(* CODESYS project ForOPC.export

Project tree, tasks and I/O mapping:
  application Application
    libraries: ; WagoAppStepper, 1.6.1.1 (WAGO)
    task PLC_Task (cyclic, interval t#50ms, priority 15) calls PLC_PRG
    DataTypes/
      data type CurveStates
      data type ForceStepStates
      data type StepperStates
      data type StiffnessTestStates
    GV/
      global variables AI_Sensors
      global variables HMI_Alm
      global variables HMI_Process
      global variables HMI_Stepper
    Program/
      Device/
        Motors/
          ForceStep/
            function block fbForceStep [ST]: METH_Direction
            program prForceStep [ST]
          Stepper/
            function block fbStepper [ST]: ACT_MoveHome, ACT_MoveToPos, METH_Direction
            program prLaserStepper_1 [ST]
            program prLaserStepper_2 [ST]
          program prMotion [ST]
        program prDevice [ST]
      IO/
        program prInToVars [ST]
      Process/
        GetCurve/
          function block fbGetCurve [ST]
          program prGetCurve_1 [ST]
          program prGetCurve_2 [ST]
        StiffnessTest/
          function block fbStiffnessTest [ST]
          program prStiffnessTest_1 [ST]
          program prStiffnessTest_2 [ST]
        program prProcess [ST]
      program prSimulation [ST]
    program PLC_PRG [ST]
    Symbols
*)

// Application/DataTypes/CurveStates

TYPE CurveStates :
(
	CS_Stop 		:= 0,
	CS_Done			:= 1,
	CS_Stopping		:= 2,
	CS_SetStep		:= 3,
	CS_WaitInitial	:= 4,
	CS_SetMeassure	:= 5,
	CS_Measuring	:= 6
);
END_TYPE

// Application/DataTypes/ForceStepStates

TYPE ForceStepStates :
(
	FS_Stop 				:= 0,
	FS_FirstRun 			:= 1,
	FS_WaitRaughApprox		:= 2,
	FS_MakeStep				:= 3,
	FS_CheckForce			:= 4,
	FS_Done					:= 5,
	FS_StartRelease			:= 6,
	FS_WaitRelease			:= 7,
	FS_MovePos				:= 8,
	FS_WaitVelicity			:= 9,
	FS_VelicityMode			:= 10,
	FS_VelicityStopping		:= 11
);
END_TYPE

// Application/DataTypes/StepperStates

TYPE StepperStates :
(
	SM_Idle 			:=0,
	SM_Homing			:=1,
	SM_Home				:=2,
	SM_SetPrm			:=3,
	SM_MovingToPos		:=4,
	SM_OnPos			:=5,
	SM_Stopping 		:=6,
	SM_Stop 			:=7
);
END_TYPE

// Application/DataTypes/StiffnessTestStates

TYPE StiffnessTestStates :
(
	ST_Proc_Stop 			:= 0,
	ST_Proc_GettingForce 	:= 1,
	ST_Proc_GettingHalfKoef	:= 2,
	ST_Proc_CalcKoef		:= 3,
	ST_Proc_GettingCurve	:= 4,
	ST_Proc_Done			:= 5,
	ST_Proc_Releasing		:= 6,
	ST_Proc_Stopping		:= 7
	
);
END_TYPE

// Application/GV/AI_Sensors

VAR_GLOBAL
	AI_Rol_1 		AT %IW1 : WORD;
	AI_Rol_2 		AT %IW2 : WORD;
	AI_Laser_1 		AT %IW3 : WORD;
	AI_Laser_2 		AT %IW4 : WORD;
	
	wCounter_1		AT %IW28 : WORD;
	wCounter_2		AT %IW30 : WORD;
	dwCounter		: DWORD;
END_VAR

// Application/GV/HMI_Alm

VAR_GLOBAL
	xResetAlm		: BOOL;
END_VAR

// Application/GV/HMI_Process

VAR_GLOBAL
	///////////////////////////   GET CURVE 1  //////////////////////
	
	xGC_Start_1: BOOL;
	wGS_State_1: CurveStates;
	
	///////////////////////////   GET CURVE 2  //////////////////////
	
	xGC_Start_2: BOOL;
	wGS_State_2: CurveStates;
	
	////////////////////////////  STIFFNESS TEST 1 /////////////////////////////
	
	xGS_StartProc_1: BOOL;
	wST_State_1: StiffnessTestStates;
	rST_Koef_1: REAL;
	wST_HalfPos_1: REAL;
	wST_HalfForce_1: REAL;
	xST_Ready_1: BOOL;
	
	////////////////////////////  STIFFNESS TEST 2 /////////////////////////////
	
	xGS_StartProc_2: BOOL;
	wST_State_2: StiffnessTestStates;
	rST_Koef_2: REAL;
	wST_HalfPos_2: REAL;
	wST_HalfForce_2: REAL;
	xST_Ready_2: BOOL;
	
	////////////////////////////  STIFFNESS TEST 3 /////////////////////////////
	
	xGS_StartProc_3: BOOL;
	wST_State_3: StiffnessTestStates;
	rST_Koef_3: REAL;
	wST_HalfPos_3: REAL;
	wST_HalfForce_3: REAL;
	xST_Ready_3: BOOL;
	
	////////////////////////////  DISTANCE /////////////////////////////
	
	rDistance_1		: REAL;
	rDistance_2		: REAL;
	rLaserDistance_1		: REAL;
	rLaserDistance_2		: REAL;
	
	xProcFinished			: BOOL;
	wProcType	: WORD;
	
END_VAR
VAR_GLOBAL RETAIN
	///////////////////////////   GET CURVE 1  //////////////////////
	
	wGC_Distance_1: WORD;
	wGC_InitialPos_1: WORD;
	wGC_EndPos_1: WORD;
	
	///////////////////////////   GET CURVE 2  //////////////////////
	
	wGC_Distance_2: WORD;
	wGC_InitialPos_2: WORD;
	wGC_EndPos_2: WORD;
	
	////////////////////////////  STIFFNESS TEST 1 /////////////////////////////
	
	rST_GetForce_1: REAL;
	rST_SetForce_1: REAL;
	wGS_WaitTillDone_1: WORD;
	
	////////////////////////////  STIFFNESS TEST 2 /////////////////////////////
	
	rST_GetForce_2: REAL;
	rST_SetForce_2: REAL;
	wGS_WaitTillDone_2: WORD;
	
END_VAR

// Application/GV/HMI_Stepper

VAR_GLOBAL
	///////////////////////    FORCE STEP    //////////////////////////////
	rFS_GetForce: REAL;	
	xFS_Start: BOOL;
	xFS_Release: BOOL;
	wFS_State: WORD;
	wFS_ActualPos: DWORD;
	xFS_JogLeft: BOOL;
	xFS_JogRight: BOOL;
	rFS_GetForce_check: REAL;	
	rFS_CycledWay:	REAL;
	rFS_LinedWay_1:	REAL;
	rFS_LinedWay_2:	REAL;
	
	
	///////////////////////////   LASER  STEP 1  //////////////////////
	xLS_MoveToPos_1: BOOL;
	xLS_MoveHome_1: BOOL;
	xLS_Stop_1: BOOL;
	wLS_GetPos_1: DINT;
	wLS_StepperState_1: WORD;
	xLS_Initilized_1: BOOL;
	rLS_RealPos_1:	REAL;
	
	///////////////////////////   LASER  STEP 2  //////////////////////
	xLS_MoveToPos_2: BOOL;
	xLS_MoveHome_2: BOOL;
	xLS_Stop_2: BOOL;
	wLS_GetPos_2: DINT;
	wLS_StepperState_2: WORD;
	xLS_Initilized_2: BOOL;
	rLS_RealPos_2:	REAL;
	
	
	
END_VAR
VAR_GLOBAL RETAIN
	
///////////////////////    FORCE STEP    //////////////////////////////
	rFS_SetForce: REAL;
	wFS_RoughApprox: WORD;
	wFS_Step: WORD;
	xFS_DirNeg: BOOL;
	rFS_Sensativity: REAL;
	wFS_SetSpeed: WORD;
	wFS_SetAcceleration: WORD;
	wFS_SetDeceleration: WORD;
	
	
///////////////////////////   LASER  STEP 1  //////////////////////	
	wLS_SetPos_1: WORD;
	wLS_SetSpeed_1: WORD;
	xLS_DirNeg_1: BOOL;
	wLS_Acceleration_1: WORD;
	wLS_Deceleration_1: WORD;
	
	///////////////////////////   LASER  STEP 2  //////////////////////	
	wLS_SetPos_2: WORD;
	wLS_SetSpeed_2: WORD;
	xLS_DirNeg_2: BOOL;
	wLS_Acceleration_2: WORD;
	wLS_Deceleration_2: WORD;
	
	
	
END_VAR

// Application/PLC_PRG
PROGRAM PLC_PRG
VAR
END_VAR

prDevice();
prProcess();
prSimulation();

END_PROGRAM

// Application/Program/Device/prDevice
PROGRAM prDevice
VAR
END_VAR

prMotion();

END_PROGRAM

// Application/Program/Device/Motors/prMotion
PROGRAM prMotion
VAR
END_VAR

prForceStep();
(*prLaserStepper_1();
prLaserStepper_2();*)

END_PROGRAM

// Application/Program/Device/Motors/ForceStep/prForceStep
PROGRAM prForceStep
VAR
	ForceStep:		fbForceStep;
	
	
	
END_VAR

ForceStep(
	rSetForce:= rFS_SetForce, 
	rGetForce:= rFS_GetForce, 
	wRoughApprox:= wFS_RoughApprox, 
	wStep:= wFS_Step, 
	xDirNeg:= xFS_DirNeg, 
	rSensativity:= rFS_Sensativity, 
	wSpeed:= wFS_SetSpeed, 
	wAcceleration:= wFS_SetAcceleration, 
	wDeceleration:= wFS_SetDeceleration, 
	I_Port:= IoConfig_Globals.Servo_Stepper_Controller_55_VDC_7_5A, 
	xStart:= xFS_Start, 
	xResetErr:= xResetAlm, 
	xRelease:= xFS_Release,
	xJogLeft:= xFS_JogLeft, 
	xJogRight:= xFS_JogRight,
	wState=> wFS_State, 
	diActualPosition=> );
	
	wFS_ActualPos:= ForceStep.diActualPosition;

END_PROGRAM

// Application/Program/Device/Motors/ForceStep/fbForceStep
FUNCTION_BLOCK fbForceStep
VAR_INPUT
	rSetForce:			REAL;
	rSetPos:			DINT;
	rGetForce:			REAL;
	wRoughApprox:		WORD;
	wStep:				WORD;
	xDirNeg:			BOOL;
	rSensativity:		REAL;
	wSpeed: 			WORD;
	wAcceleration: 		WORD;
	wDeceleration: 		WORD;
	I_Port: 			WagoAppStepper.WagoTypesModule_75x_67x.I_Module_75x_67x;
END_VAR
VAR_IN_OUT
	xStart:				BOOL;
	xResetErr:			BOOL;
	xRelease:			BOOL;
	xJogLeft:			BOOL;
	xJogRight:			BOOL;
END_VAR
VAR_OUTPUT
	wState:				ForceStepStates;
	diActualPosition: 	DINT;
END_VAR
VAR
	rtStart:			R_TRIG;
	ftStart:			F_TRIG;
	ftRelease:			F_TRIG;
	ControlBasic:		WagoAppStepper.FbStepperControlBasic;
	xEnable: 			BOOL;
	eJobType: 			WagoAppStepper.eMode;
	xTriggerStart: 		BOOL;
	xTriggerErrorReset: BOOL;
	xStop: 				BOOL;
	
	
	diPosition: 		DINT;
	iSpeed: 			INT;
	xJobFinished: 		BOOL;
	xBusy: 				BOOL;
	xError: 			BOOL;
	oStatus: 			WagoAppStepper.WagoSysErrorBase.FbResult;
	eErrorCodes: 		WagoAppStepper.eStatus;
	diRoughDistance:	DINT;
	rCompareForce:		REAL;
	rDirection:			INT;
	rtRelease:			R_TRIG;
	rtJogLeft:			R_TRIG;
	rtJogright:			R_TRIG;
	
END_VAR

VAR RETAIN
	diRetainPos: DINT;
END_VAR

rtStart(CLK:=xStart);
ftStart(CLK:=xStart);
rtRelease(CLK:=xRelease);
ftRelease(CLK:=xRelease);
rtJogLeft(CLK:=xJogLeft);
rtJogright(CLK:=xJogRight);

IF (ftStart.Q OR ftRelease.Q)AND (NOT (wState = FS_Done)) THEN
	xStop			:= TRUE;
	xTriggerStart	:= FALSE;
	xRelease		:= FALSE;	
	wState:=FS_Stop;
END_IF

IF rtRelease.Q THEN
	xStop			:=TRUE;
	xTriggerStart	:= FALSE;
	xJogLeft		:= FALSE;
	xJogRight		:= FALSE;
	wState			:=FS_StartRelease;
END_IF

IF (rtJogLeft.Q OR rtJogright.Q) AND (NOT(wState = FS_Stop OR wState = FS_Done)) THEN
	xJogLeft		:= FALSE;
	xJogRight		:= FALSE;
END_IF


CASE wState OF
	
		FS_Stop, FS_Done:
		
		
				IF rtStart.Q THEN
					diRoughDistance		:= 0;
					xStop				:=FALSE;
					rCompareForce		:= (rSetForce/100)* wRoughApprox;
					METH_Direction(xDirNeg:= xDirNeg);
					IF rSetPos = 0 THEN
						wState			:= FS_FirstRun;
					ELSE
						xEnable			:= TRUE;
						eJobType		:= MoveRelative;
						diPosition		:= rSetPos;
						iSpeed			:= wSpeed;
						xTriggerStart	:= TRUE;
						wState			:= FS_MovePos;
					END_IF					
				END_IF
				
				IF xJogLeft OR xJogRight THEN
					xEnable			:= TRUE;
					xStop			:=FALSE;
					eJobType		:= VelocityControl;
					METH_Direction(xDirNeg:= xJogLeft);
					iSpeed			:= (TO_INT(wSpeed)) * rDirection;
					xTriggerStart	:= TRUE;
					wState			:= FS_WaitVelicity;
				END_IF
					
		
		FS_FirstRun:
		
				xEnable			:= TRUE;
				eJobType		:= MoveRelative;
				diPosition		:= 200000 * rDirection;
				iSpeed			:= wSpeed;
				xTriggerStart	:=TRUE;
				wState			:= FS_WaitRaughApprox;
				
				
		FS_WaitRaughApprox:
		
				IF rGetForce > rCompareForce THEN
					xStop	:=TRUE;
					wState	:= FS_MakeStep;
				END_IF
				
		
		FS_MakeStep:
				
		
				IF xJobFinished THEN
					xStop			:=FALSE;
					diPosition		:= wStep * rDirection;
					xTriggerStart	:=TRUE;
					wState			:= FS_CheckForce;
				END_IF
				
				
		FS_CheckForce:
		
				
				IF xJobFinished THEN
					IF (rGetForce < rSetForce + rSensativity) AND (rGetForce > rSetForce - rSensativity) THEN
						xStart	:=FALSE;
						wState	:= FS_Done;
					ELSIF rGetForce < rSetForce - rSensativity THEN
						METH_Direction(xDirNeg:= xDirNeg);
						wState	:= FS_MakeStep;
					ELSIF rGetForce > rSetForce + rSensativity THEN
						METH_Direction(xDirNeg:= NOT xDirNeg);
						wState	:= FS_MakeStep;
					END_IF
				END_IF
				
		FS_StartRelease:
		
				IF xJobFinished THEN
					xStop			:=FALSE;
					METH_Direction(xDirNeg:= NOT xDirNeg);
					xEnable			:= TRUE;
					eJobType		:= MoveRelative;
					diPosition		:= 200000 * rDirection;
					iSpeed			:= wSpeed;
					xTriggerStart	:=TRUE;
					wState			:= FS_WaitRelease;
				END_IF
				
		FS_WaitRelease:
		
				IF rGetForce < rSensativity THEN
					xStart:= FALSE;
					xStop			:= TRUE;
					xTriggerStart	:= FALSE;
					xRelease		:= FALSE;	
					wState:=FS_Stop;
				END_IF
				
				
		FS_MovePos:
		
				IF xJobFinished THEN
					wState	:= FS_Done;
				END_IF
				
				
		FS_WaitVelicity:
		
				IF NOT xTriggerStart THEN
					wState	:= FS_VelicityMode;
				END_IF
				
				
		FS_VelicityMode:
		
		
				IF rtJogLeft.Q OR rtJogright.Q THEN
					xJogRight		:=rtJogright.Q;
					xJogLeft		:=rtJogLeft.Q;
					METH_Direction(xDirNeg:= xJogLeft);
					iSpeed			:= (TO_INT(wSpeed)) * rDirection;
					xTriggerStart	:= TRUE;
				END_IF
		
				IF NOT (xJogLeft OR xJogRight) THEN
					iSpeed			:= 0;
					xTriggerStart	:= TRUE;
					wState			:= FS_VelicityStopping;
				END_IF
				
				
		FS_VelicityStopping:
		
				IF ControlBasic.iActualSpeed = 0 AND (NOT xTriggerStart) THEN
					wState			:= FS_Stop;
				END_IF
				

END_CASE





ControlBasic(
	xEnable:= xEnable, 
	I_Port:= I_Port, 
	eJobType:= eJobType, 
	xDirPos:= NOT xDirNeg, 
	xDirNeg:= xDirNeg, 
	iSpeed:= iSpeed, 
	wAcceleration:= wAcceleration, 
	wDeceleration:= wDeceleration, 
	diPosition:= diPosition, 
	xTriggerStart:= xTriggerStart, 
	xTriggerErrorReset:= xTriggerErrorReset, 
	xStop:= xStop, 
	xJobFinished=> xJobFinished, 
	xBusy=> xBusy, 
	xError=> xError, 
	oStatus=> oStatus, 
	eErrorCodes=> eErrorCodes, 
	diActualPosition=> diActualPosition, 
	iActualSpeed=> , 
	xMailboxActive=> , 
	xResetWarning=> );

METHOD METH_Direction
VAR_INPUT
	xDirNeg:	BOOL;
END_VAR
IF xDirNeg THEN
	rDirection:= -1;
ELSE
	rDirection:= 1;
END_IF
END_METHOD

END_FUNCTION_BLOCK

// Application/Program/Device/Motors/Stepper/prLaserStepper_1
PROGRAM prLaserStepper_1
VAR
	LaserStepper	:	fbStepper;
	xMoveRelative	: 	BOOL;
	wRatio			: 	WORD:=10;
	
		
END_VAR

LaserStepper(
	diSetPos:= wLS_SetPos_1 * wRatio, 
	xMoveRelative:= xMoveRelative, 
	iSetSpeed:= wLS_SetSpeed_1 * wRatio, 
	xDirNeg:= xLS_DirNeg_1, 
	wAcceleration:= wLS_Acceleration_1, 
	wDeceleration:= wLS_Deceleration_1, 
	I_Port:= IoConfig_Globals.Servo_Stepper_Controller_55_VDC_7_5A_1, 
	xMoveToPos:= xLS_MoveToPos_1, 
	xMoveHome:= xLS_MoveHome_1, 
	xStop:= xLS_Stop_1, 
	diGetPos=> , 
	xInitilized=> xLS_Initilized_1, 
	wStepperState=> wLS_StepperState_1);
	
	wLS_GetPos_1:=LaserStepper.diGetPos/wRatio;

END_PROGRAM

// Application/Program/Device/Motors/Stepper/fbStepper
FUNCTION_BLOCK fbStepper
VAR_INPUT
	diSetPos:			DINT;
	xMoveRelative:		BOOL;
	iSetSpeed:			INT;
	xDirNeg:			BOOL;
	wAcceleration: 		WORD;
	wDeceleration: 		WORD;
	I_Port: 			WagoAppStepper.WagoTypesModule_75x_67x.I_Module_75x_67x;
END_VAR
VAR_IN_OUT
	xMoveToPos:			BOOL;
	xMoveHome:			BOOL;
	xStop:				BOOL;
END_VAR
VAR_OUTPUT
	diGetPos:			DINT;
	xInitilized:		BOOL;
	wStepperState:		StepperStates;
END_VAR
VAR
	rtMoveToPos:		R_TRIG;
	rtMoveHome:			R_TRIG;
	rtStop:				R_TRIG;
	ControlBasic:		WagoAppStepper.FbStepperControlBasic;
	xEnable: 			BOOL;
	eJobType: 			WagoAppStepper.eMode;
	xTriggerStart: 		BOOL;
	xTriggerErrorReset: BOOL;
	iSpeed: 			INT;
	
	diPosition: 		DINT;
	
	xJobFinished: 		BOOL;
	xBusy: 				BOOL;
	xError: 			BOOL;
	oStatus: 			WagoAppStepper.WagoSysErrorBase.FbResult;
	eErrorCodes: 		WagoAppStepper.eStatus;
	diRoughDistance:	DINT;
	rCompareForce:		REAL;
	rDirection:			INT;
	iActualSpeed: INT;
	SetPosition:WagoAppStepper.FbSetPosition;
	xSetZeroPos: BOOL;
	xHome: BOOL;
	rtHome:	R_TRIG;
	xStopLoc: BOOL;
END_VAR

rtMoveToPos(CLK:=xMoveToPos);
rtMoveHome(CLK:=xMoveHome);
rtStop(CLK:=xStop);

IF rtMoveHome.Q THEN	
	wStepperState:= SM_Idle;
END_IF

IF rtStop.Q THEN
	xStopLoc		:= TRUE;
	xMoveToPos		:= FALSE;
	xMoveHome		:= FALSE;
	wStepperState	:= SM_Stopping;
END_IF


CASE wStepperState OF
	
		
			SM_Idle:
			
								
				IF rtMoveToPos.Q OR rtMoveHome.Q THEN
					ACT_MoveHome();					
				END_IF
				
				IF xBusy AND iActualSpeed <> 0 AND (xMoveToPos OR xMoveHome) THEN
					wStepperState	:= SM_Homing;
				END_IF
				
				
			SM_Homing:
			
				IF xBusy AND iActualSpeed = 0 THEN
					xStopLoc:= TRUE;
				END_IF
				IF NOT xBusy THEN
					xStopLoc	:= FALSE;
					xSetZeroPos	:= TRUE;
				END_IF
				rtHome(CLK:=xHome);
				IF rtHome.Q THEN
					xSetZeroPos		:= FALSE;
					xStopLoc		:= FALSE;
					xInitilized		:= TRUE;
					xMoveHome		:= FALSE;
					wStepperState	:= SM_Home;
				END_IF
				
				
			SM_Home, SM_OnPos, SM_Stop:
			
				IF xMoveToPos THEN
					ACT_MoveToPos();
				END_IF
				
				
			SM_SetPrm:
			
				IF xBusy THEN
					xTriggerStart	:=FALSE;
					wStepperState	:= SM_MovingToPos;
				END_IF
				
				
			SM_MovingToPos:
			
				IF xJobFinished THEN
					xMoveToPos		:=FALSE;
					wStepperState	:= SM_OnPos;
				END_IF
				
				
			SM_Stopping:
			
				IF NOT xBusy THEN
					xStopLoc		:= FALSE;
					xStop			:= FALSE;
					IF xInitilized THEN
						wStepperState	:= SM_Stop;
					ELSE
						wStepperState	:= SM_Idle;
					END_IF
				END_IF
				
END_CASE



ControlBasic(
	xEnable:= xEnable, 
	I_Port:= I_Port, 
	eJobType:= eJobType, 
	xDirPos:= NOT xDirNeg, 
	xDirNeg:= xDirNeg, 
	iSpeed:= iSetSpeed, 
	wAcceleration:= wAcceleration, 
	wDeceleration:= wDeceleration, 
	diPosition:= diPosition, 
	xTriggerStart:= xTriggerStart, 
	xTriggerErrorReset:= xTriggerErrorReset, 
	xStop:= xStopLoc, 
	xJobFinished=> xJobFinished, 
	xBusy=> xBusy, 
	xError=> xError, 
	oStatus=> oStatus, 
	eErrorCodes=> eErrorCodes, 
	diActualPosition=> diGetPos, 
	iActualSpeed=> iActualSpeed, 
	xMailboxActive=> , 
	xResetWarning=> );
	
SetPosition(
	xExecute:= xSetZeroPos, 
	I_Port:= I_Port, 
	diPosition:= 60, 
	xDone=> xHome, 
	xBusy=> , 
	xError=> , 
	oStatus=> );

ACTION ACT_MoveHome:
	METH_Direction(xDirNeg:= NOT xDirNeg);
	xEnable			:= TRUE;
	xStopLoc		:= FALSE;
	eJobType		:= MoveRelative;
	diPosition		:= 200000 * rDirection;
	xTriggerStart	:=TRUE;
END_ACTION

ACTION ACT_MoveToPos:
	METH_Direction(xDirNeg:= xDirNeg);
	xStopLoc			:= FALSE;
	xEnable			:= TRUE;					
	eJobType		:= MoveAbsolute;
	diPosition		:= diSetPos;
	xTriggerStart	:=TRUE;
	wStepperState	:= SM_SetPrm;
END_ACTION

METHOD METH_Direction
VAR_INPUT
	xDirNeg:	BOOL;
END_VAR
IF xDirNeg THEN
	rDirection:= -1;
ELSE
	rDirection:= 1;
END_IF
END_METHOD

END_FUNCTION_BLOCK

// Application/Program/Device/Motors/Stepper/prLaserStepper_2
PROGRAM prLaserStepper_2
VAR
	LaserStepper	:	fbStepper;
	xMoveRelative	: 	BOOL;
	wRatio			: 	WORD:=10;
END_VAR

LaserStepper(
	diSetPos:= wLS_SetPos_2 * wRatio, 
	xMoveRelative:= xMoveRelative, 
	iSetSpeed:= wLS_SetSpeed_2 * wRatio, 
	xDirNeg:= xLS_DirNeg_2, 
	wAcceleration:= wLS_Acceleration_2, 
	wDeceleration:= wLS_Deceleration_2, 
	I_Port:= IoConfig_Globals.Servo_Stepper_Controller_55_VDC_7_5A_2, 
	xMoveToPos:= xLS_MoveToPos_2, 
	xMoveHome:= xLS_MoveHome_2, 
	xStop:= xLS_Stop_2, 
	diGetPos=> , 
	xInitilized=> xLS_Initilized_2, 
	wStepperState=> wLS_StepperState_2);
	
	wLS_GetPos_2:=LaserStepper.diGetPos/wRatio;

END_PROGRAM

// Application/Program/Process/prProcess
PROGRAM prProcess
VAR
END_VAR

prGetCurve_1();
prGetCurve_2();
prStiffnessTest_1();
prStiffnessTest_2();
IF xProcFinished THEN
	xProcFinished:= FALSE;
END_IF

END_PROGRAM

// Application/Program/Process/GetCurve/prGetCurve_1
PROGRAM prGetCurve_1
VAR
	GetCurve	: fbGetCurve;	
END_VAR

GetCurve(
	diDistance:= wGC_Distance_1, 
	wStepperState:= wLS_StepperState_1, 
	xInitilized:= xLS_Initilized_1, 
	wInitialPos:= wGC_InitialPos_1, 
	wEndPos:= wGC_EndPos_1, 
	xStart:= xGC_Start_1, 
	xMovePos:= xLS_MoveToPos_1, 
	xStopStep:= xLS_Stop_1, 
	wSetPos:= wLS_SetPos_1, 
	wState=> wGS_State_1);

END_PROGRAM

// Application/Program/Process/GetCurve/fbGetCurve
FUNCTION_BLOCK fbGetCurve
VAR_INPUT
	diDistance		: DINT;
	wStepperState	: StepperStates;
	xInitilized		: BOOL;
	wInitialPos		: WORD;
	wEndPos			: WORD;
END_VAR
VAR_IN_OUT
	xStart			: BOOL;
	xMovePos		: BOOL;
	xStopStep		: BOOL;
	wSetPos			: WORD;
END_VAR
VAR_OUTPUT
	wState			: CurveStates;	
END_VAR
VAR
	rtStart			: R_TRIG;
	ftStart			: F_TRIG;
END_VAR

rtStart(CLK:= xStart);
ftStart(CLK:= xStart);

IF ftStart.Q AND (NOT (wState = CS_Done))THEN
	xStopStep:= TRUE;
	wState:= CS_Stopping;
END_IF


CASE wState OF
	

		CS_Stop, CS_Done:
		
			IF xStart THEN
				xMovePos	:= TRUE;
				wSetPos		:= wInitialPos;
				wState		:= CS_SetStep;
			END_IF
			
			
		CS_SetStep:
		
			IF wStepperState = SM_MovingToPos THEN
				wState		:= CS_WaitInitial;
			END_IF
			
		CS_WaitInitial:
		
			IF wStepperState = SM_OnPos THEN
				xMovePos	:= TRUE;
				wSetPos		:= wEndPos;
				wState		:= CS_SetMeassure;
			END_IF
			
		CS_SetMeassure:
		
			IF wStepperState = SM_MovingToPos THEN
				wState		:= CS_Measuring;
			END_IF 
				
		CS_Measuring:
		
			IF wStepperState = SM_OnPos THEN
				xStart		:= FALSE;
				wState		:= CS_Done;
			END_IF
	


END_CASE

END_FUNCTION_BLOCK

// Application/Program/Process/GetCurve/prGetCurve_2
PROGRAM prGetCurve_2
VAR
	GetCurve	: fbGetCurve;	
END_VAR

GetCurve(
	diDistance:= wGC_Distance_2, 
	wStepperState:= wLS_StepperState_2, 
	xInitilized:= xLS_Initilized_2, 
	wInitialPos:= wGC_InitialPos_2, 
	wEndPos:= wGC_EndPos_2, 
	xStart:= xGC_Start_2, 
	xMovePos:= xLS_MoveToPos_2, 
	xStopStep:= xLS_Stop_2, 
	wSetPos:= wLS_SetPos_2, 
	wState=> wGS_State_2);

END_PROGRAM

// Application/Program/Process/StiffnessTest/prStiffnessTest_1
PROGRAM prStiffnessTest_1
VAR
	StiffnessTest: fbStiffnessTest;	
END_VAR

StiffnessTest(
	xReady:= xST_Ready_1, 
	rGetForce:= rST_GetForce_1, 
	rSetForce:= rST_SetForce_1, 
	wGetPos:= wFS_ActualPos, 
	wFS_State:= wFS_State, 
	wCSState:= wGS_State_1, 
	wWaitTillDone:= wGS_WaitTillDone_1, 
	xStartProc:= xGS_StartProc_1, 
	xStartForce:= xFS_Start, 
	xStartCurve:= xGC_Start_1, 
	xReleaseForce:= xFS_Release, 
	wState=> wST_State_1, 
	rKoef=> rST_Koef_1, 
	wHalfPos=> );
	
xST_Ready_1:= wProcType <> 0;
wST_HalfPos_1:= StiffnessTest.wHalfPos;

END_PROGRAM

// Application/Program/Process/StiffnessTest/fbStiffnessTest
FUNCTION_BLOCK fbStiffnessTest
VAR_INPUT
	xReady			: BOOL;
	rGetForce		: REAL;
	rSetForce		: REAL;
	wGetPos			: DWORD;
	wFS_State		: ForceStepStates;
	wCSState		: CurveStates;
	wWaitTillDone	: WORD;
END_VAR
VAR_IN_OUT
	xStartProc		: BOOL;
	xStartForce		: BOOL;
	xStartCurve		: BOOL;
	xReleaseForce	: BOOL;
END_VAR
VAR_OUTPUT
	wState			: StiffnessTestStates;
	rKoef			: REAL;
	wHalfPos		: DWORD;
END_VAR
VAR
	rtStart			: R_TRIG;
	ftStart			: F_TRIG;
	rtGetHalf		: R_TRIG;
	tnWaitTillDone	: TON;	
	HalfPos			: DWORD;
	StartPos		: DWORD;
END_VAR

rtStart(CLK:= xStartProc);
ftStart(CLK:= xStartProc);

IF ftStart.Q AND (NOT(wState = ST_Proc_Done)) THEN
	xStartForce		:= FALSE;
	xStartCurve		:= FALSE;
	xReleaseForce	:= FALSE;
	tnWaitTillDone(IN:= FALSE); 
	wState			:= ST_Proc_Stopping;
END_IF


CASE wState OF
	

		ST_Proc_Stop, ST_Proc_Done:
		
				IF xStartProc THEN
					xStartForce := TRUE;
					StartPos	:= wGetPos;
					wState		:= ST_Proc_GettingForce;
				END_IF
				
				
		ST_Proc_GettingForce:
		
		
				rtGetHalf(CLK:= rGetForce > (rSetForce * 0.5));
				IF rtGetHalf.Q THEN
					wHalfPos := wGetPos - StartPos;
				END_IF
				
				IF wFS_State = FS_Done AND rGetForce > (rSetForce * 0.5) THEN
					wState	:= ST_Proc_CalcKoef;
				END_IF
				
				
		ST_Proc_CalcKoef:
		
				tnWaitTillDone(IN:= wFS_State = FS_Done, PT:= TO_TIME(wWaitTillDone * 1000));
				IF tnWaitTillDone.Q THEN
					tnWaitTillDone(IN:= FALSE); 
					rKoef 		:= (0.5 * rGetForce)/(wGetPos - wHalfPos);
					xStartCurve := TRUE;
					wState		:= ST_Proc_GettingCurve;
				END_IF
				
				
		ST_Proc_GettingCurve:
		
		
				tnWaitTillDone(IN:= wCSState = CS_Done, PT:= TO_TIME(wWaitTillDone * 1000)); 
				IF tnWaitTillDone.Q THEN
					tnWaitTillDone(IN:= FALSE); 
					xStartCurve 	:= FALSE;
					xReleaseForce	:= TRUE;
					wState			:=ST_Proc_Releasing;
				END_IF
				

		ST_Proc_Releasing:
				

				IF 	wFS_State = FS_Stop THEN
					xStartProc 	:= FALSE;
					wState		:=ST_Proc_Done;
				END_IF
				
		ST_Proc_Stopping:
		
				IF (wFS_State = FS_Stop OR wFS_State = FS_Done) AND (wCSState = CS_Stop OR wCSState = CS_Done) THEN
					wState		:=ST_Proc_Stop;
				END_IF

END_CASE

END_FUNCTION_BLOCK

// Application/Program/Process/StiffnessTest/prStiffnessTest_2
PROGRAM prStiffnessTest_2
VAR
	StiffnessTest: fbStiffnessTest;	
END_VAR

StiffnessTest(
	xReady:= xST_Ready_2, 
	rGetForce:= rST_GetForce_2, 
	rSetForce:= rST_SetForce_2, 
	wGetPos:= wFS_ActualPos, 
	wFS_State:= wFS_State, 
	wCSState:= wGS_State_2, 
	wWaitTillDone:= wGS_WaitTillDone_2, 
	xStartProc:= xGS_StartProc_2, 
	xStartForce:= xFS_Start, 
	xStartCurve:= xGC_Start_2, 
	xReleaseForce:= xFS_Release, 
	wState=> wST_State_2, 
	rKoef=> rST_Koef_2, 
	wHalfPos=> wST_HalfPos_2);
	
xST_Ready_2:= wProcType <> 0;
wST_HalfPos_2:= StiffnessTest.wHalfPos;

END_PROGRAM

// Application/Program/prSimulation
PROGRAM prSimulation
VAR
END_VAR

rFS_GetForce := wFS_ActualPos;
rFS_GetForce_check := wFS_ActualPos;
rFS_CycledWay := wFS_ActualPos / 2;

END_PROGRAM

// Application/Program/IO/prInToVars
PROGRAM prInToVars
VAR
	k_1: REAL;
	k_2: REAL;
	k_3: REAL;
	k_4: REAL;
END_VAR

(*rDistance_1 := TO_REAL(AI_Rol_1) * k_1;*)
rDistance_2 := TO_REAL(AI_Rol_2) * k_2;
rLaserDistance_1 := TO_REAL(AI_Laser_1) * k_3;
rLaserDistance_2 := TO_REAL(AI_Laser_2) * k_4;

END_PROGRAM
